// TIA Portal V20 export
DATA_BLOCK "DB_Inst"   // DB6
// stored: InstanceOfName FB_Lad, InstanceOfType FB
"FB_Lad"
   // VAR_INPUT
   //    Start : Bool;
   // END_VAR
BEGIN
END_DATA_BLOCK
